FUNCTION_BLOCK StopAerate2 (* Basic Function Block Type *)
  (* Standard: 61499-2 *)
  (* Version 0.0, 7/16/2026, Schneider Electric, Template *)
  PACKAGE SE.Nereda;
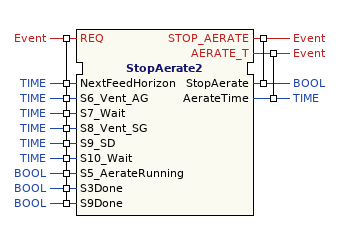
  EVENT_INPUT
    REQ WITH NextFeedHorizon, S6_Vent_AG, S7_Wait, S8_Vent_SG, S5_AerateRunning, S3Done, S9Done, S9_SD, S10_Wait; (* Normal Execution Request *)
  END_EVENT
  EVENT_OUTPUT
    STOP_AERATE WITH StopAerate; (* Execution Confirmation *)
    AERATE_T WITH AerateTime;
  END_EVENT
  VAR_INPUT
    NextFeedHorizon : TIME;
    S6_Vent_AG : TIME;
    S7_Wait : TIME;
    S8_Vent_SG : TIME;
    S9_SD : TIME;
    S10_Wait : TIME;
    S5_AerateRunning : BOOL;
    S3Done : BOOL;
    S9Done : BOOL;
  END_VAR
  VAR_OUTPUT
    StopAerate : BOOL;
    AerateTime : TIME;
  END_VAR
  VAR
    VentAGTime : REAL;
    VentSGTime : REAL;
    SDTime : REAL;
    WaitTime1 : REAL;
    WaitTime2 : REAL;
    InNextFeedHorizon : REAL;
    SumState : REAL;
  END_VAR
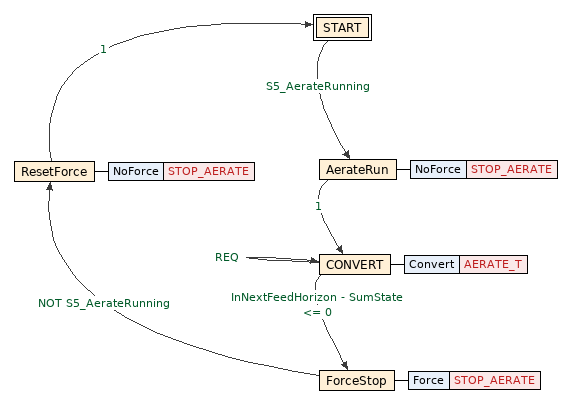
  EC_STATES
    START; (* Initial State *)
    AerateRun : NoForce -> STOP_AERATE;
    ForceStop : Force -> STOP_AERATE;
    ResetForce : NoForce -> STOP_AERATE;
    CONVERT : Convert -> AERATE_T;
  END_STATES
  EC_TRANSITIONS
    START TO AerateRun := S5_AerateRunning;
    CONVERT TO ForceStop := InNextFeedHorizon - SumState <= 0;
    ForceStop TO ResetForce := NOT S5_AerateRunning;
    ResetForce TO START := 1;
    AerateRun TO CONVERT := 1;
    CONVERT TO CONVERT := REQ;
  END_TRANSITIONS
  ALGORITHM NoForce IN ST:
;
StopAerate := FALSE;
  END_ALGORITHM
  ALGORITHM Force IN ST:
;
StopAerate := TRUE;
  END_ALGORITHM
  ALGORITHM Convert IN ST:
VentAGTime := TIME_TO_REAL(S6_Vent_AG / 1000);
VentSGTime := TIME_TO_REAL(S8_Vent_SG / 1000);
SDTime := TIME_TO_REAL(S9_SD / 1000);
WaitTime1 := TIME_TO_REAL(S7_Wait / 1000);
WaitTime2 := TIME_TO_REAL(S10_Wait / 1000);
InNextFeedHorizon := TIME_TO_REAL(NextFeedHorizon / 1000);

IF S3Done THEN
	SumState := VentAGTime + VentSGTime + WaitTime1 + WaitTime2;
ELSE
	SumState := VentAGTime + VentSGTime + WaitTime1 + WaitTime2 + SDTime;
END_IF;

AerateTime := REAL_TO_TIME((InNextFeedHorizon - SumState) * 1000);
  END_ALGORITHM
END_FUNCTION_BLOCK
